// TIA Portal V16 export
// export: Created 2022-09-29T17:53:39.3578115Z, ExportSetting WithDefaults, DisplayName Totally Integrated Automation Portal, DisplayVersion V16, DisplayName TIA Portal Version Control Interface, DisplayVersion V16, DisplayName TIA Portal Openness, DisplayVersion V16, DisplayName STEP 7 Professional, DisplayVersion V16, DisplayName STEP 7 Safety, DisplayVersion V16, DisplayName WinCC Advanced, DisplayVersion V16
ORGANIZATION_BLOCK "Main"   // OB1, LAD, ProgramCycle
TITLE = "Main Program Sweep (Cycle)"
{ S7_Optimized_Access := 'TRUE' }
VERSION : 0.1
// stored: AutoNumber true, IsIECCheckEnabled false, SetENOAutomatically false
BEGIN

REGION Network 1: Alimentação ao processo
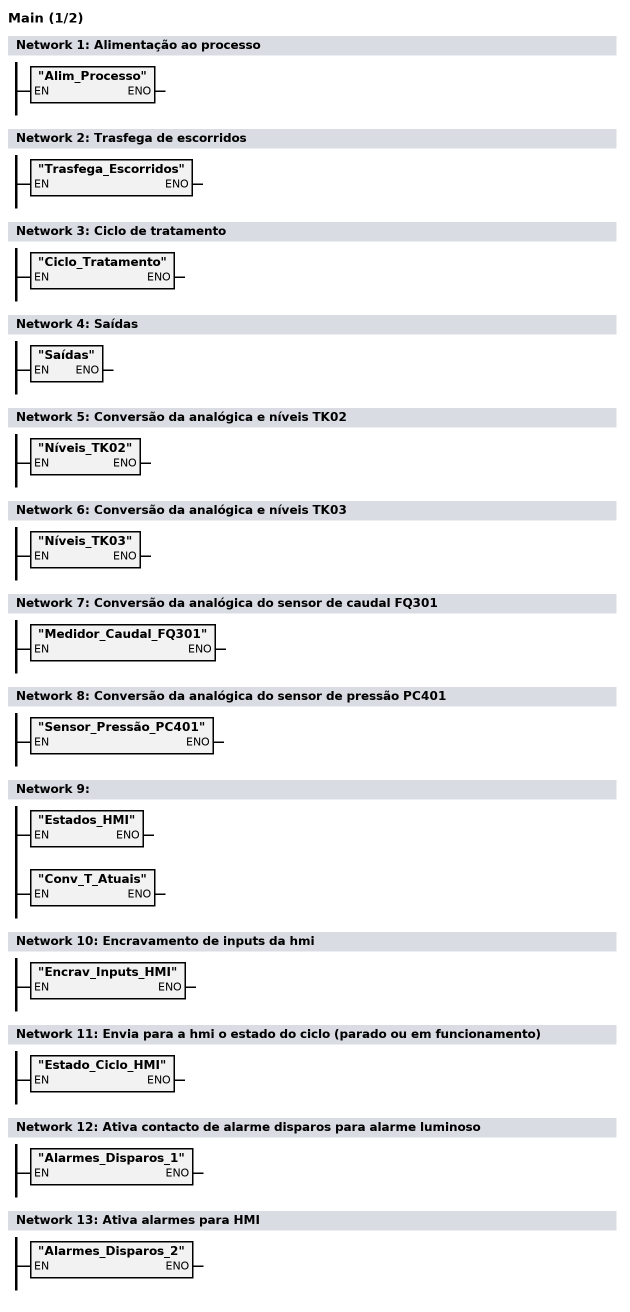
   RUNG wire#powerrail
      "Alim_Processo"()
   END_RUNG
   // the same network as SCL:
   "Alim_Processo"();
END_REGION

REGION Network 2: Trasfega de escorridos
   RUNG wire#powerrail
      "Trasfega_Escorridos"()
   END_RUNG
   // the same network as SCL:
   "Trasfega_Escorridos"();
END_REGION

REGION Network 3: Ciclo de tratamento
   RUNG wire#powerrail
      "Ciclo_Tratamento"()
   END_RUNG
   // the same network as SCL:
   "Ciclo_Tratamento"();
END_REGION

REGION Network 4: Saídas
   RUNG wire#powerrail
      "Saídas"()
   END_RUNG
   // the same network as SCL:
   "Saídas"();
END_REGION

REGION Network 5: Conversão da analógica e níveis TK02
   RUNG wire#powerrail
      "Níveis_TK02"()
   END_RUNG
   // the same network as SCL:
   "Níveis_TK02"();
END_REGION

REGION Network 6: Conversão da analógica e níveis TK03
   RUNG wire#powerrail
      "Níveis_TK03"()
   END_RUNG
   // the same network as SCL:
   "Níveis_TK03"();
END_REGION

REGION Network 7: Conversão da analógica do sensor de caudal FQ301
   RUNG wire#powerrail
      "Medidor_Caudal_FQ301"()
   END_RUNG
   // the same network as SCL:
   "Medidor_Caudal_FQ301"();
END_REGION

REGION Network 8: Conversão da analógica do sensor de pressão PC401
   RUNG wire#powerrail
      "Sensor_Pressão_PC401"()
   END_RUNG
   // the same network as SCL:
   "Sensor_Pressão_PC401"();
END_REGION

REGION Network 9
   RUNG wire#powerrail
      "Estados_HMI"()
   END_RUNG
   RUNG wire#powerrail
      "Conv_T_Atuais"()
   END_RUNG
   // the same network as SCL:
   "Estados_HMI"();
   "Conv_T_Atuais"();
END_REGION

REGION Network 10: Encravamento de inputs da hmi
   RUNG wire#powerrail
      "Encrav_Inputs_HMI"()
   END_RUNG
   // the same network as SCL:
   "Encrav_Inputs_HMI"();
END_REGION

REGION Network 11: Envia para a hmi o estado do ciclo (parado ou em funcionamento)
   RUNG wire#powerrail
      "Estado_Ciclo_HMI"()
   END_RUNG
   // the same network as SCL:
   "Estado_Ciclo_HMI"();
END_REGION

REGION Network 12: Ativa contacto de alarme disparos para alarme luminoso
   RUNG wire#powerrail
      "Alarmes_Disparos_1"()
   END_RUNG
   // the same network as SCL:
   "Alarmes_Disparos_1"();
END_REGION

REGION Network 13: Ativa alarmes para HMI
   RUNG wire#powerrail
      "Alarmes_Disparos_2"()
   END_RUNG
   // the same network as SCL:
   "Alarmes_Disparos_2"();
END_REGION

REGION Network 14: Alarme XV102 (não abriu/não fechou)
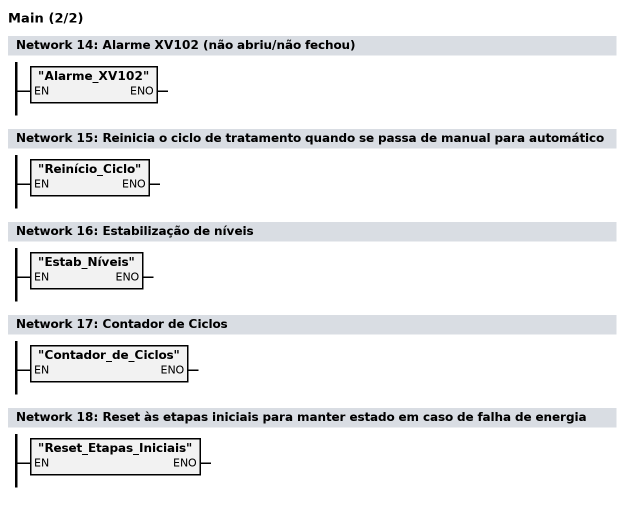
   RUNG wire#powerrail
      "Alarme_XV102"()
   END_RUNG
   // the same network as SCL:
   "Alarme_XV102"();
END_REGION

REGION Network 15: Reinicia o ciclo de tratamento quando se passa de manual para automático
   RUNG wire#powerrail
      "Reinício_Ciclo"()
   END_RUNG
   // the same network as SCL:
   "Reinício_Ciclo"();
END_REGION

REGION Network 16: Estabilização de níveis
   RUNG wire#powerrail
      "Estab_Níveis"()
   END_RUNG
   // the same network as SCL:
   "Estab_Níveis"();
END_REGION

REGION Network 17: Contador de Ciclos
   RUNG wire#powerrail
      "Contador_de_Ciclos"()
   END_RUNG
   // the same network as SCL:
   "Contador_de_Ciclos"();
END_REGION

REGION Network 18: Reset às etapas iniciais para manter estado em caso de falha de energia
   RUNG wire#powerrail
      "Reset_Etapas_Iniciais"()
   END_RUNG
   // the same network as SCL:
   "Reset_Etapas_Iniciais"();
END_REGION
END_ORGANIZATION_BLOCK
